{attribute 'linkalways'} 
{attribute 'no_explicit_call' := 'This FB is a CLASS and must be accessed using methods or properties'}
{attribute 'enable_dynamic_creation'}
FUNCTION_BLOCK FINAL SUB_INT EXTENDS Node
VAR
	in1 : _INT(0);
	in2 : _INT(0);
	out : _INT(0);
END_VAR

METHOD PUBLIC Clone : I_Node
VAR
	pNode : POINTER TO SUB_INT;
END_VAR
pNode := __NEW(SUB_INT);
Clone := pNode^;
END_METHOD

METHOD FB_init : BOOL
VAR_INPUT
	bInitRetains : BOOL; // if TRUE, the retain variables are initialized (warm start / cold start)
	bInCopyCode : BOOL;  // if TRUE, the instance afterwards gets moved into the copy code (online change)
END_VAR
AddInput('in1',THIS^.in1);
AddInput('in2',THIS^.in2);
AddOutput('out', THIS^.out);
END_METHOD

METHOD PROTECTED OnExecute
VAR
END_VAR
out.Value := in1.Value - in2.Value;
END_METHOD

END_FUNCTION_BLOCK

(* stored: Version 1.1.0.1, ProductVersion 3.1.4024.15
   POU SUB_INT: Id {4b1d61d3-0001-4616-b018-1cf18a6412a2}, SpecialFunc None
   Folder Constructor: Id {59e97730-c71b-4343-ae6c-816e6e34e9d8}
   Method Clone: Id {140102b9-f799-406a-92cd-a02093a8e14f}
   Method FB_init: Id {cdbb6e18-3a6b-47d9-a909-3920a6c42710}
   Method OnExecute: Id {5894d45d-976c-4cad-8a69-6ee055a45d3e} *)
